{attribute 'qualified_only'}
VAR_GLOBAL
	fJoystickNormalizedY 		: LREAL; 
	fJoystickNormalizedX 		: LREAL; 
	fJoystickNormalizedZ 		: LREAL; 
	fYokeNormalizedFeedback 	: LREAL; 
	fPressureWinchA 	 		: LREAL; 
	fPressureWinchB 	 		: LREAL; 
	fPressureSupply 	 		: LREAL; 
	fPressureReturn 	 		: LREAL; 
	fWinchEncoderPosition 		: LREAL;
	fPayLoadPosition 			: LREAL;
	fDeltaPMotor 				: LREAL;
END_VAR

(* stored: Version 1.1.0.1
   GVL G_Scaled_values: Id {4ff3b0b3-7afb-45b2-8b55-d797c734f296} *)
